Yaskawa INFORM job: GO-TO-STATION-1-FRONT.JBI

/JOB
//NAME GO-TO-STATION-1-FRONT
//POS
///NPOS 2,0,0,1,0,0
///TOOL 0
///POSTYPE PULSE
///PULSE
C00000=-124951,-185456,-1458,-3200,-135233,158604
C00001=-107423,-36358,10351,68056,-126377,117727
P00000=0,-222014,-26224,0,-132993,0
//INST
///DATE 2018/08/27 13:34
///ATTR SC,RW
///GROUP1 RB1
NOP
MOVJ P0000 VJ=50.00
'*****
SETREG MREG#(1) 1
MOVJ C00000 VJ=25.00
'*****
SETREG MREG#(1) 10
MOVJ C00001 VJ=25.00
'*****
SETREG MREG#(1) 11
END
